// TIA Portal V20 export
FUNCTION "FC_INPUT_MAP" : Void   // FC101, LAD
{ S7_Optimized_Access := 'TRUE' }
// stored: AutoNumber false, SetENOAutomatically false
   VAR_TEMP
      LOOP : Int;
      Value : Byte;
   END_VAR
BEGIN

REGION Network 1 (SCL): INPUT900BYTE
   FOR #LOOP := 0 TO 900 BY 1 DO
       #Value := PEEK(area := 16#81, dbNumber := 0, byteOffset := #LOOP);
       POKE(area:=16#84,dbNumber:=40, byteOffset:=#LOOP,value:=#Value);
   END_FOR;
END_REGION
END_FUNCTION
